Omron CX-Programmer project NewProject (CX-Programmer 9.70)

# PLC NewPLC1: CP1E E20

## Global symbols (name address type ; comment)
0.00 BOOL  ; input

## Program NewProgram1 (cyclic task 0)

### Section Section1

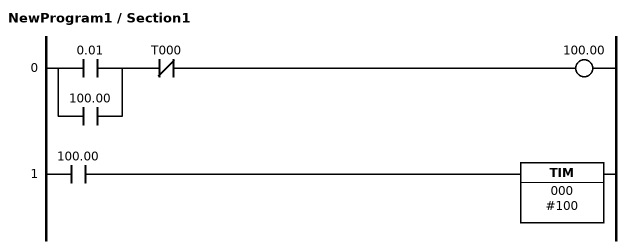
; rung 0
LD 0.01
OR 100.00
ANDNOT T000
OUT 100.00
; rung 1
LD 100.00
TIM 000 #100

### Section END
; rung 0
END(001)